TYPE ValueType : __SYSTEM.TYPE_CLASS; END_TYPE

(* stored: Version 1.1.0.1, ProductVersion 3.1.4024.15
   DUT ValueType: Id {4aa9d4f1-e1bf-48ab-ac3b-e0269e0f158d} *)
